VAR_GLOBAL CONSTANT
	MaxNrofMessages: UINT:= 30;
END_VAR

VAR_GLOBAL
	
END_VAR

(* stored: Version 1.1.0.1, ProductVersion 3.1.4026.18
   GVL GVL: Id {c749aa94-77ca-4d45-832d-ac09e2bd2780} *)
